{attribute 'qualified_only'}
{attribute 'strict'}
TYPE LevitationSystemSTM :
(
	Idling,
	Stationary,
	Transitioning,
	HoldingAirGap,
	TransitioningToZero
);
END_TYPE

(* stored: Version 1.1.0.1, ProductVersion 3.1.4024.12
   DUT LevitationSystemSTM: Id {52699997-7127-4c93-8117-00d4c3457941} *)
